INTERFACE I_CoeAccess EXTENDS I_Base

PROPERTY CoE : I_CoeDevice
GET
END_GET
END_PROPERTY

END_INTERFACE

(* stored: Version 1.1.0.1, ProductVersion 3.1.4026.18
   Itf I_CoeAccess: Id {a3087a82-f1ad-437d-af74-916da87ee094}
   Property CoE: Id {49b1e6de-fe14-42f7-862a-864aaf734f1f}
   Get Get: Id {af59799e-005b-4f81-841d-41529f0311ce} *)
